Fanuc KAREL source: kd00026.KL

-- PROVISIONAL review KL for V940-1; original PC SHA256 f71651f612a126bccd8f8ce2cb2e083e31540b57e0b8bd1fe943c00c10aefc09
-- Incomplete behavior may be omitted. Consult companion uncertainty JSON. Do not deploy.
PROGRAM KD00026
%NOLOCKGROUP
VAR
  I : INTEGER
  J : INTEGER
  B : BOOLEAN
  R : REAL
  S : STRING[80]
BEGIN
  -- V9_ZERO_TABLE_METADATA_HINT layout=0001; no indexed target words; source/name/runtime held
  -- UNRESOLVED_PC offsets 5-24; opcodes 9D,81,18,9D,1B,9D,12,22,9D,13,04
  -- UNRESOLVED_PC offsets 29-33; opcodes 7F
END KD00026
